PROGRAM Step_8_Outfeed
VAR
// ------------triggers-----------------	
rtPullRope_8 : R_TRIG;



//--------safety---------------------
LocalSafety_8: BOOL;
	
	
	
	
END_VAR



//----------------------Safety--------------------

LocalSafety_8 := OutFeedConveyorMMP;


//---------------------Defaults-------------------


rtPullRope_8(CLK := OutfeedRopePull);


// Stop button or lost permissive or lost local safety → go to IDLE immediately
IF CycleStopPB OR NOT Permissive THEN
    Step5_State := 0; // IDLE
END_IF	



// ----------------------------------- Manual override (when AutoMode = FALSE) ---------------------------------------
IF NOT AutoMode THEN
    OutFeedConveyorFWD := FALSE;
	
    IF Permissive AND LocalSafety_8 THEN
        // Only run FWD if REV jog is NOT pressed
        IF OutFeedConveyorFWD THEN
            GradingVFD2FWD := TRUE;
		ELSE
			OutFeedConveyorFWD := FALSE;
        END_IF

    END_IF;

    RETURN;
END_IF



//--------------------------AutoMode---------------------------------------------------------------------------
CASE Step8_State OF

0: // Stopped  


OutFeedConveyorFWD := FALSE;


IF CycleStartPB OR rtPullRope_8.Q THEN
    Step5_State := 5; // IDLE
END_IF	


5: // Running/Standby
   
OutFeedConveyorFWD := TRUE;

IF rtPullRope_8.Q THEN
	Step5_State := 0;

END_IF





END_CASE;

END_PROGRAM

(* stored: Version 1.1.0.1
   POU Step_8_Outfeed: Id {164f23e4-e886-4aca-984d-e8e72a062bab}, SpecialFunc None *)
